PROGRAM TEST_UNIT_MASTER
VAR
	fbVirtual : RunUnitIndexerMaster(ptBlock:= ADR(GVL.LOCAL_UNIT_CONTEXTS[4]),
									 ptUpstream:=0);
	fbMaster : RunUnitIndexerMaster(ptBlock:= ADR(GVL.LOCAL_UNIT_CONTEXTS[3]),
									ptUpstream := ADR(fbVirtual));
END_VAR

fbVirtual.ProxyMode(netID:= '10.221.24.70.1.1',port :=851);
fbMaster();

END_PROGRAM

(* stored: Version 1.1.0.1, ProductVersion 3.1.4020.12
   POU TEST_UNIT_MASTER: Id {e52701ab-3d6a-4aa0-bffd-71a5234ebd5a}, SpecialFunc None *)
